# EPICS autosave request: norhofLN2/norhofLN2_positions.req
$(P):TIMETOOFF
$(P):TIMETOSLEEP
$(P):TIMETOWASH_FROMOFF
$(P):TIMETOWASH_FROMSLEEP
$(P):TIMETOWASH_FROMSTANDBY
$(P):WASH_COUNT
$(P):WASH_COUNT_TOTAL
$(P):WASH_PRES
